PROGRAM MAIN
VAR
	opcData1: INT;
	bInit : BOOL;
END_VAR

opcData1 := 7;

END_PROGRAM

(* stored: Version 1.1.0.1
   POU MAIN: Id {28be77c9-9914-0795-3937-baecd3c16a40}, SpecialFunc None *)
